TYPE ST_BoxCorner : 
	STRUCT 
		PointXTime : LREAL; 
		PointYValue : LREAL; 
	END_STRUCT
END_TYPE

(* stored: Version 1.1.0.1, ProductVersion 3.1.4024.11
   DUT ST_BoxCorner: Id {53c510b1-abda-0c02-0c89-a18443e417b2} *)
